// TIA Portal V17 export
// export: Created 2024-09-02T12:50:32.299616Z, ExportSetting WithDefaults, DisplayName Totally Integrated Automation Portal, DisplayVersion V17, DisplayName TIA Portal Openness, DisplayVersion V17, DisplayName TIA Portal Version Control Interface, DisplayVersion V17, DisplayName STEP 7 Professional, DisplayVersion V17, DisplayName STEP 7 Safety, DisplayVersion V17, DisplayName WinCC Professional, DisplayVersion V17
TYPE "TypeSKS_Feeder_Unit"
// stored: IsFailsafeCompliant false
   STRUCT
      "A" : Struct
         on : Bool;
         off : Bool;
         Part_Out : Bool;
      END_STRUCT;
      H : Struct
         on : Bool;
         off : Bool;
         Part_Out : Bool;
      END_STRUCT;
      Status : Struct
         Part_insite : Bool;
         Part_in_way : Bool;
      END_STRUCT;
   END_STRUCT;
END_TYPE
